{attribute 'linkalways'} 
{attribute 'no_explicit_call' := 'This FB is a CLASS and must be accessed using methods or properties'}
{attribute 'enable_dynamic_creation'}
FUNCTION_BLOCK FINAL Node_UDINT_TO_LREAL EXTENDS Node
VAR
	in : _UDINT(0);
	out : _LREAL(0.0);
	success : _BOOL(FALSE);
END_VAR

METHOD PUBLIC  Clone : I_Node
VAR
	pNode : POINTER TO Node_UDINT_TO_LREAL;
END_VAR
pNode := __NEW(Node_UDINT_TO_LREAL);
Clone := pNode^;
END_METHOD

METHOD FB_init : BOOL
VAR_INPUT
	bInitRetains : BOOL; // if TRUE, the retain variables are initialized (warm start / cold start)
	bInCopyCode : BOOL;  // if TRUE, the instance afterwards gets moved into the copy code (online change)
END_VAR
AddParameter('in', in);
AddOutput('out', out);
AddOutput('success', success);

this^.Metadatum.AddBoolAsMetadata('deprecated', true);
END_METHOD

METHOD PROTECTED OnExecute
VAR
END_VAR
success.Value := TryConvert_UDINT_TO_LREAL(in.Value, out.Value);
END_METHOD

END_FUNCTION_BLOCK

(* stored: Version 1.1.0.1, ProductVersion 3.1.4026.18
   POU Node_UDINT_TO_LREAL: Id {a9a6bbb3-7c3c-0995-19c4-65000583a378}, SpecialFunc None
   Folder Constructor: Id {ea8fef28-635b-0f80-0a58-26c754b97aeb}
   Method Clone: Id {b5d900d2-2cec-09dc-33bb-c9ec118d5272}
   Method FB_init: Id {f28729b3-97c5-069d-0125-4ada655d4530}
   Method OnExecute: Id {e5b0edbe-73f5-0873-251a-33bc85d9d54c} *)
